METHOD PUBLIC ShiftRange : BOOL
VAR_INPUT
	StartPos	: INT;
	EndPos 		: INT;
END_VAR
VAR
	i : INT;
	N : INT := 0;
END_VAR
IF(StartPos < EndPos AND EndPos <= ArraySize) THEN
	N := EndPos - StartPos - 1;
	FOR i:= 0 TO N DO
		MEMCPY(ADR(DataRepository[EndPos-i]), ADR(DataRepository[EndPos-i-1]), SIZEOF(stShiftData));
	END_FOR;
ELSE
	; //Error;
END_IF;

// Clear start position data array
MEMSET(ADR(DataRepository[StartPos]), 16#00, SIZEOF(stShiftData));
END_METHOD

METHOD Update : BOOL
VAR_INPUT
END_VAR
// TODO: GraphQL mutation with FIFO
END_METHOD

END_FUNCTION_BLOCK

// ---- FBs/FB_PneumaticActuator_2EV.TcPOU
FUNCTION_BLOCK FB_PneumaticActuator_2EV
VAR_INPUT
	I_bEnable					: BOOL;
	I_bCmdFwd					: BOOL;					// Comando avanti
	I_bCmdBwd					: BOOL;					// Comando indietro
	I_eReadyPos					: eReadyPos := Bwd;		// Posizione iniziale di fuori ingombro per start ciclo 0=indietro, 1=avanti
	I_bSensorFwd				: BOOL;					// Sensore avanti
	I_bSensorBwd				: BOOL;					// Sensore indietro
	I_bCmdReset					: BOOL;					// Reset allarmi
	I_bAirPresence				: BOOL;					// Presenza aria nel circuito - Abilitazione comandi
	I_bManualMode				: BOOL;					// Modo manuale
	I_bEvMonostable				: BOOL;
	I_tTimeoutFwd				: TIME := T#0S;			// Timeout movimento avanti
	I_tTimeoutBwd				: TIME := T#0S;			// Timeout movimento indietro
	I_tDelaySensorFwd			: TIME := T#0S;			// Ritardo sul sensore avanti
	I_tDelaySensorBwd			: TIME := T#0S;			// Ritardo sul sensore indietro
	I_tWarningFwd				: TIME := T#0S;			// Warning movimento avanti  
	I_tWarningBwd				: TIME := T#0S;			// Warning movimento indietro
END_VAR

VAR_OUTPUT
	Q_bActuatorFwd				: BOOL := FALSE;		// Comando avanti
	Q_bActuatorBwd				: BOOL := FALSE;		// Comando indietro
	Q_bTimeoutFwd				: BOOL := FALSE;		// Timeout avanti attivo
	Q_bTimeoutBwd				: BOOL := FALSE;		// Timeout indietro attivo
	Q_bWarningFwd				: BOOL := FALSE;		// Warning avanti attivo
	Q_bWarningBwd				: BOOL := FALSE;		// Warning indietro attivo
	Q_bSensorBroken				: BOOL := FALSE;		// Timeout entrambi sensori attivi
	Q_bDelaySensorFwd			: BOOL := FALSE;		// Stato sensore avanti ritardato
	Q_bDelaySensorBwd			: BOOL := FALSE;		// Stato sensore indietro ritardato
	Q_tElapsedTimeFwd			: UINT := 0;			// Durata movimento avanti
	Q_tElapsedTimeBwd			: UINT := 0;			// Durata movimento indietro
	Q_tLastFwd					: UINT := 0;			// Durata ultimo movimento avanti
	Q_tLastBwd					: UINT := 0;			// Durata ultimo movimento indietro
	Q_bReadyPos					: BOOL := FALSE;		// In posizione iniziale di fuori ingombro
	Q_eStatus					: eEV_Status := eEV_Status.NotUsed; // Descrizione stato funzione
END_VAR

VAR
	_TON_TimerFwd				: TON;
	_TON_TimerBwd				: TON;
	_TON_WarningFwd				: TON;
	_TON_WarningBwd				: TON;
	_TON_TimerSensorBroken		: TON;
	_TON_DelaySensorFwd			: TON;	
	_TON_DelaySensorBwd			: TON;
END_VAR

_TON_DelaySensorFwd(IN := I_bSensorFwd, PT := I_tDelaySensorFwd, Q => Q_bDelaySensorFwd);					
_TON_DelaySensorBwd(IN := I_bSensorBwd, PT := I_tDelaySensorBwd, Q => Q_bDelaySensorBwd);

_TON_TimerFwd(IN := Q_bActuatorFwd AND NOT I_bSensorFwd AND I_bAirPresence);					
_TON_TimerBwd(IN := Q_bActuatorBwd AND NOT I_bSensorBwd AND I_bAirPresence);
												
IF I_bEnable THEN
	IF I_bManualMode THEN
		// Logica di movimento in indietro
		IF I_bCmdBwd THEN
			Q_bActuatorBwd := TRUE;
			Q_bActuatorFwd := FALSE;
			Q_eStatus := eEV_Status.MovingBackward;
		ELSIF NOT I_bEvMonostable AND NOT I_bCmdBwd THEN
			Q_bActuatorBwd := FALSE;
		END_IF
		// Logica di movimento in avanti
		IF I_bCmdFwd THEN
			Q_bActuatorFwd := TRUE;
			Q_bActuatorBwd := FALSE;
			Q_eStatus := eEV_Status.MovingForward;  
		ELSIF NOT I_bEvMonostable AND NOT I_bCmdFwd THEN
			Q_bActuatorFwd := FALSE;
		END_IF
	ELSE
		// Logica di movimento in avanti
		IF I_bCmdFwd AND NOT I_bSensorFwd THEN
		    Q_bActuatorFwd := TRUE;          
		    Q_bActuatorBwd := FALSE;         
		    Q_eStatus := eEV_Status.MovingForward;   
		ELSIF I_bSensorFwd AND NOT I_bEvMonostable THEN
		    Q_bActuatorFwd := FALSE;         
		END_IF
	
		// Logica di movimento indietro
		IF I_bCmdBwd AND NOT I_bSensorBwd THEN
		    Q_bActuatorBwd := TRUE;          				
		    Q_bActuatorFwd := FALSE;         				
		    Q_eStatus := eEV_Status.MovingBackward;	
		ELSIF I_bSensorBwd AND NOT I_bEvMonostable THEN
		    Q_bActuatorBwd := FALSE;         				
		END_IF
	END_IF	
END_IF

// Status
IF (Q_eStatus = eEV_Status.MovingBackward AND I_bSensorBwd) OR (Q_eStatus = eEV_Status.MovingForward AND I_bSensorFwd) THEN
	Q_eStatus := eEV_Status.MoveCompleted;
END_IF	

// Condizione di sicurezza: evitare comandi simultanei
IF I_bCmdFwd AND I_bCmdBwd THEN
    Q_bActuatorFwd := FALSE;	
    Q_bActuatorBwd := FALSE;    
END_IF
		
// Ready Position
IF(((I_eReadyPos = Bwd AND I_bSensorBwd) OR (I_eReadyPos = Fwd AND I_bSensorFwd)) AND NOT Q_bSensorBroken AND NOT Q_bTimeoutBwd AND NOT Q_bTimeoutFwd) THEN
	Q_bReadyPos := TRUE;
ELSE
	Q_bReadyPos := FALSE;
END_IF

// Elapsed Time	
Q_tElapsedTimeBwd := TIME_TO_UINT(_TON_TimerBwd.ET);
Q_tElapsedTimeFwd := TIME_TO_UINT(_TON_TimerFwd.ET);
IF I_bSensorFwd THEN
	Q_tLastFwd := Q_tElapsedTimeFwd;
ELSIF I_bSensorBwd THEN
	Q_tLastBwd := Q_tElapsedTimeBwd;
END_IF	

// Timeout
_TON_TimerBwd.PT := SEL(I_tTimeoutBwd = T#0S, I_tTimeoutBwd, T#99S);
_TON_TimerFwd.PT := SEL(I_tTimeoutFwd = T#0S, I_tTimeoutFwd, T#99S);
IF(_TON_TimerFwd.Q AND (I_tTimeoutFwd > T#0S)) AND I_bAirPresence THEN
	Q_bTimeoutFwd 	:= TRUE;
END_IF
IF(_TON_TimerBwd.Q AND (I_tTimeoutBwd > T#0S)) AND I_bAirPresence THEN
	Q_bTimeoutBwd 	:= TRUE;
END_IF

// Warning
_TON_WarningFwd(IN := Q_eStatus = eEV_Status.MovingForward AND NOT I_bSensorFwd AND I_bAirPresence, PT := I_tWarningFwd);					
_TON_WarningBwd(IN := Q_eStatus = eEV_Status.MovingBackward AND NOT I_bSensorBwd AND I_bAirPresence, PT := I_tWarningBwd);
IF I_bAirPresence THEN
	IF _TON_WarningFwd.Q AND (I_tWarningFwd > T#0S) THEN
		Q_bWarningFwd 	:= TRUE;
	ELSE
		Q_bWarningFwd 	:= FALSE;
	END_IF
	IF _TON_WarningBwd.Q AND (I_tWarningBwd > T#0S) THEN
		Q_bWarningBwd 	:= TRUE;
	ELSE
		Q_bWarningBwd 	:= FALSE;
	END_IF
END_IF

// Error - Sensor broken
_TON_TimerSensorBroken(PT := T#100MS, Q => Q_bSensorBroken);
IF I_bSensorFwd AND I_bSensorBwd  THEN
	_TON_TimerSensorBroken.IN := TRUE;
ELSE
	_TON_TimerSensorBroken.IN := FALSE;
END_IF

// Error management
IF Q_bTimeoutBwd OR Q_bTimeoutFwd OR Q_bSensorBroken THEN
	IF NOT Q_bSensorBroken THEN
		Q_eStatus := eEV_Status.Timeout;
	ELSE
		Q_eStatus := eEV_Status.Error;
	END_IF
END_IF

// Reset function
IF(I_bCmdReset) THEN
	Q_bTimeoutFwd 		:= FALSE;
	Q_bTimeoutBwd 		:= FALSE;
	Q_bSensorBroken		:= FALSE;
END_IF

END_FUNCTION_BLOCK

// ---- FBs/LaserMarker - LASIT/FC_Check_STX.TcPOU
FUNCTION FC_Check_STX : BOOL
VAR_INPUT
	I_sString : REFERENCE TO T_MaxString;
END_VAR
VAR
	stringPos	: INT;
END_VAR

stringPos := FIND(I_sString, STX);
IF stringPos <> 0 THEN
	I_sString := MID(I_sString, LEN(I_sString), stringPos+1);
	FC_Check_STX := TRUE;
ELSE
	FC_Check_STX := FALSE;
END_IF

END_FUNCTION

// ---- FCs/FC_EnumSnakeCaseToString.TcPOU
FUNCTION FC_EnumSnakeCaseToString : STRING
VAR_INPUT
	I_String	: T_MaxString; // Use TO_STRING(eNum) to convert the input enum. For empty string set enum = eNull
END_VAR
VAR
	pos			: INT;				
END_VAR

IF I_String <> 'eNull' THEN
	IF LEFT(I_String, 1) = 'e' THEN
		I_String := DELETE(I_String, 1, 1);
	END_IF
	pos := FIND(I_String, '_');
	WHILE pos <> 0 DO
		I_String := REPLACE(I_String, ' ', 1, pos);
		pos := FIND(I_String, '_');
	END_WHILE
	FC_EnumSnakeCaseToString := I_String;
ELSE
	FC_EnumSnakeCaseToString := '';
END_IF

END_FUNCTION

// ---- FCs/FC_MarkingLayoutSelection.TcPOU
FUNCTION FC_MarkingLayoutSelection : STRING(243)
VAR_INPUT
	Source	: eMarkingLayoutSource;
	Text	: STRING;
	MarkingCode : STRING(243);
	ProductName : STRING(243);
END_VAR

IF Source = eMarkingLayoutSource.ProductName THEN
	FC_MarkingLayoutSelection := ProductName;
ELSIF Source = eMarkingLayoutSource.FreeText THEN
	FC_MarkingLayoutSelection := Text;
ELSE
	FC_MarkingLayoutSelection := MarkingCode;
END_IF

END_FUNCTION

// ---- FCs/FC_OvrManagement.TcPOU
FUNCTION FC_OvrManagement : UINT
VAR_INPUT
	X_min 			: UINT;
    X_max 			: UINT;
    Y_min 			: UINT;
    Y_max 			: UINT;
	Counter			: UINT;
	SetCounterDone 	: BOOL;
END_VAR
VAR_OUTPUT
	SetCounte 		: BOOL;
	SetCounteValue 	: UINT;
END_VAR

IF NOT SetCounterDone THEN
	IF Counter < X_min THEN
		SetCounteValue := X_min;
		SetCounte := TRUE;
	ELSIF Counter > X_max THEN
		SetCounteValue := X_max;
		SetCounte := TRUE;
	ELSE
		FC_OvrManagement := (((Counter - X_min) * (Y_max - Y_min)) / (X_max - X_min) + Y_min);
	END_IF
ELSIF SetCounte THEN
	SetCounte := FALSE;
END_IF

END_FUNCTION

// ---- FCs/FC_PMCAlarmToBoolArray.TcPOU
FUNCTION FC_PMCAlarmToBoolArray : BOOL
VAR_INPUT
	RegA : POINTER TO BYTE;
END_VAR
VAR_OUTPUT
	AlarmList : ARRAY[0..CNC.NUM_MAX_STATION_ALARMS-1] OF BOOL;
END_VAR
VAR
	i : LWORD;
	j : DINT;
	reg: BYTE;
END_VAR

FOR i:= 0 TO 9 DO
	FOR j := 0 TO 7 DO
        AlarmList[(i*8) + j] := TO_BOOL(PBYTE_TO_BYTE((RegA+i)) AND SHL(1,j));
    END_FOR
END_FOR

END_FUNCTION

// ---- FCs/FC_PMCWarningToBoolArray.TcPOU
FUNCTION FC_PMCWarningToBoolArray : BOOL
VAR_INPUT
	RegA : POINTER TO BYTE;
END_VAR
VAR_OUTPUT
	WarningList : ARRAY[0..CNC.NUM_MAX_STATION_WARNINGS-1] OF BOOL;
END_VAR
VAR
	i : LWORD;
	j : DINT;
	reg: BYTE;
END_VAR

FOR i:= 0 TO 9 DO
	FOR j := 0 TO 7 DO
        WarningList[(i*8) + j] := TO_BOOL(PBYTE_TO_BYTE((RegA+i)) AND SHL(1,j));
    END_FOR
END_FOR

END_FUNCTION

// ---- FCs/FC_ProductStatusDatabase.TcPOU
FUNCTION FC_ProductStatusDatabase : eDbPiecesStatus
VAR_INPUT
	In					: STRING(50);
END_VAR

IF In = 'Completed' THEN
	FC_ProductStatusDatabase := eDbPiecesStatus.Completed;
ELSIF In = 'Scrap' THEN
	FC_ProductStatusDatabase := eDbPiecesStatus.Scrap;
ELSIF In = 'Processing' THEN
	FC_ProductStatusDatabase := eDbPiecesStatus.Processing;
ELSIF In = 'Fetched' THEN
	FC_ProductStatusDatabase := eDbPiecesStatus.Fetched;
ELSIF In = 'Undefined' THEN
	FC_ProductStatusDatabase := eDbPiecesStatus.Undefined;
ELSE
	FC_ProductStatusDatabase := eDbPiecesStatus.Undefined;
END_IF

END_FUNCTION

// ---- FCs/FC_SetPartProgramNameByID.TcPOU
FUNCTION FC_SetPartProgramNameByID : STRING
VAR_INPUT
	Id : LINT;
END_VAR
VAR
	sId : STRING;
	str : STRING(9) := 'O00000000';
END_VAR


sId := LINT_TO_STRING(id);
FC_SetPartProgramNameByID := CONCAT(LEFT(str, 9 - LEN(sId)), sId);

END_FUNCTION

// ---- FCs/FC_ToBoolArray.TcPOU
FUNCTION FC_ToBoolArray
VAR_INPUT
	RegSource : POINTER TO BYTE;
	RegDest	  : POINTER TO BOOL;
	Size : UINT;
END_VAR
VAR
	i 	: LWORD;
	j 	: DINT;
	reg : BYTE;
END_VAR

FOR i:=0 TO Size-1 DO
	FOR j:= 0 TO 7 DO
		RegDest^ := TO_BOOL(PBYTE_TO_BYTE((RegSource+i)) AND SHL (1,j));	
		RegDest := RegDest+1;
	END_FOR
END_FOR

END_FUNCTION

// ---- FCs/FC_ToByte.TcPOU
FUNCTION FC_ToByte : BOOL
VAR_INPUT
	RegSource : POINTER TO BOOL;
	RegDest	  : POINTER TO BYTE;
	Size : UINT;
END_VAR
VAR
	i 	: DINT;
	j   : DINT;
	bitIndex : INT;
	byteIndex : INT;
	temp : BYTE;
END_VAR

FOR i:=0 TO size-1 BY 8 DO
	temp := 0;
	FOR j:= 0 TO 7 DO
		IF RegSource[i+j] THEN
			temp := temp OR (SHL(1,j));
		END_IF
	END_FOR
	RegDest^ := temp;
	RegDest:=RegDest+1;
END_FOR

END_FUNCTION

// ---- FCs/FC_WIDP_TO_PPNAME.TcPOU
FUNCTION FC_WIDP_TO_PPNAME : STRING
VAR_INPUT
	WindP					: STRING;
END_VAR
VAR
	i				: INT;
	tempPPINT 		: INT;
	tempPPString	: STRING;
END_VAR

tempPPINT := LEN(WindP);
tempPPString := WindP;
IF tempPPINT < 8 THEN
	FOR i := 0 TO 7-tempPPINT DO
		tempPPString := CONCAT('0', tempPPString);
	END_FOR
END_IF
FC_WIDP_TO_PPNAME := tempPPString;

END_FUNCTION

// ---- FCs/Inc.TcPOU
FUNCTION Inc
VAR_INPUT
	In : POINTER TO DINT;
END_VAR

In^ := In^ + 1;

END_FUNCTION

// ---- FCs/Print.TcPOU
FUNCTION Print : BOOL
VAR_INPUT
	Text : T_MaxString;
	Arg	: T_MaxString;
END_VAR

ADSLOGSTR(ADSLOG_MSGTYPE_LOG, CONCAT(Text, '%s'), Arg);

END_FUNCTION

// ---- POUs/Database.TcPOU
PROGRAM Database
VAR
	i : UDINT;
	fbMSSQLCommandEvt 			: ARRAY[0..DB.MAX_NUMBER_ST] OF FB_SQLCommandEvt(sNetID := '', tTimeout := T#10S);
	fbMSSQLStoreProcedureEvt	: ARRAY[0..DB.MAX_NUMBER_ST] OF FB_SQLStoredProcedureEvt(sNetID := '', tTimeout := T#10S);
	tempfbMSSQLStoreProcedureEvt : ARRAY[0..DB.MAX_NUMBER_ST] OF POINTER TO FB_SQLStoredProcedureEvt; 
	fbMSSQLResult				: ARRAY[0..DB.MAX_NUMBER_ST] OF FB_SQLResultEvt(sNetID := '', tTimeout := T#10S);
	
	spUpdatePartLocationsAndProcessingDataParameters		: DUT_UpdatePartLocationsAndProcessingData;
	stParameterProcessingDataForHMI		: DUT_ProcessingDataForHMI;
	
	resetProcessinData						: BOOL;
	
	RTRIG_ProcessingDataExecute	 : R_TRIG;
	RTRIG_ShiftManTrigger0to1	 : R_TRIG;
	FTRIG_Running : F_TRIG;
	RTRIG_MachineEmpty	 : R_TRIG;
	RTRIG_ProcessingDataDoneError	: R_TRIG;
	
	ProcessingDataTrigger : BOOL;
	RTRIG_LogModeStateEventExecute	: R_TRIG;
	RTRIG_LogModeStateEventDoneOrError	: R_TRIG;
	LogModeStateEventTrigger	: BOOL;
	MemFirstCycle	: BOOL := FALSE;
	TempString	: STRING;
	SystemTimeSecStr	: STRING(2);
	TON_DelayLogModeStateEventTrigger : TON;
	RTRIG_GetSettingRepositoryExecute	: R_TRIG;
	RTRIG_GetSettingRepositoryDoneError	: R_TRIG;
	TON_MSSQL_spGetProcessingDataForHMIBusy : TON;
	memReq : BOOL;
	RTRIG_MesManualExecute	: R_TRIG;
	RTRIG_MesManualDoneError	: R_TRIG;
	myPeriod : TON;
	RTRIG_MyExe : R_TRIG;
	RTRIG_MyDone : R_TRIG;
	RTRIG_MyError : R_TRIG;
	myTime	: TIME := T#1S;
	myStart : BOOL;
	myVar : BOOL;
	myEnableConnection : BOOL;
	myConnected : ARRAY[1..5] OF BOOL;
END_VAR

IF _TaskInfo[MAIN.fbGetCurTaskIndex.index].FirstCycle THEN
	MemFirstCycle := TRUE;
END_IF
TempString := DT_TO_STRING(G.SystemTime);
SystemTimeSecStr := RIGHT(TempString, 2);
IF SystemTimeSecStr = '00' AND MemFirstCycle AND PRG_MSSQL_InitConnection.Connected THEN
	TON_DelayLogModeStateEventTrigger.IN := TRUE;
END_IF
TON_DelayLogModeStateEventTrigger(PT := T#500MS);
IF SystemTimeSecStr <> '00' AND LogModeStateEventTrigger AND NOT TON_DelayLogModeStateEventTrigger.IN THEN
 	LogModeStateEventTrigger := FALSE;
END_IF
IF TON_DelayLogModeStateEventTrigger.Q THEN
	LogModeStateEventTrigger := TRUE;
	TON_DelayLogModeStateEventTrigger.IN := FALSE;
END_IF



FOR i := 0 TO DB.MAX_NUMBER_ST DO
	tempfbMSSQLStoreProcedureEvt[i] := ADR(fbMSSQLStoreProcedureEvt[i]);
END_FOR

A_MSSQL();
A_MSSQL_ProcessingData();
Test();

ACTION A_MSSQL:
PRG_MSSQL_InitConnection(
						Enable			:=,
						DBID 			:= 1, 
						tRetryConn 	:= T#10S, 
						pSQLCommand1 	:= ADR(fbMSSQLCommandEvt[0]),
						pSQLCommand2 	:= ADR(fbMSSQLCommandEvt[1]),
						pSQLCommand3 	:= ADR(fbMSSQLCommandEvt[2]),
						pSQLCommand4 	:= ADR(fbMSSQLCommandEvt[3]),
						pSQLStoredProcedureEvt := tempfbMSSQLStoreProcedureEvt
						);
						 
PRG_MSSQL_spGetNextPartPLCData( Enable := PRG_MSSQL_InitConnection.Connected,
								OtherSPBusy := PRG_MSSQL_UpdatePartLocationsAndProcessingData.Busy OR PRG_MSSQL_UpdatePartLocationsAndProcessingData.Execute,
								fbSQLStoredProcedure := fbMSSQLStoreProcedureEvt[8],
								fbSQLResult := fbMSSQLResult[8],
								stPLCData := DB.stPLCData);
								
								
PRG_MSSQL_UpdatePartLocationsAndProcessingData(	Enable := PRG_MSSQL_InitConnection.Connected,
												fbSQLStoredProcedure := fbMSSQLStoreProcedureEvt[9],
												fbSQLResult := fbMSSQLResult[9],
												stProcessingData := DB.stProcessingData,
												Parameters := spUpdatePartLocationsAndProcessingDataParameters);
									
PRG_MSSQL_spGetProcessingDataForHMI( Enable := PRG_MSSQL_InitConnection.Connected,
									 Parameters := stParameterProcessingDataForHMI,
						  			 fbSQLStoredProcedure := fbMSSQLStoreProcedureEvt[10],
						  			 fbSQLResult := fbMSSQLResult[10],
									 ProcessingHMIDataLocation	=> DB.ProcessingHMIDataLocation,
									 ProcessingHMIDataViewData	=> DB.ProcessingHMIDataViewData); 
									 
IF G.MachineEmpty THEN
	MEMSET(ADR(DB.ProcessingHMIDataViewData), 0, SIZEOF(DB.ProcessingHMIDataViewData));
	MEMSET(ADR(DB.ProcessingHMIDataLocation), 0, SIZEOF(DB.ProcessingHMIDataLocation));
ELSE
	DB.ProcessingHMIDataLocation := PRG_MSSQL_spGetProcessingDataForHMI.ProcessingHMIDataLocation;
	DB.ProcessingHMIDataViewData := PRG_MSSQL_spGetProcessingDataForHMI.ProcessingHMIDataViewData;	
END_IF	

PRG_MSSQL_spCMD_AbortProduction(Enable := PRG_MSSQL_InitConnection.Connected,
						  	fbSQLStoredProcedure := fbMSSQLStoreProcedureEvt[36],
						  	fbSQLResult := fbMSSQLResult[36]);

//////////////// gestione PRG_MSSQL_spLogModeStateEvent ////////////////
RTRIG_LogModeStateEventExecute(CLK := G.OperatingModeOld <> HMI.Out.Header.OperatingMode OR G.MachineStateOld <> HMI.Out.Header.MachineState OR LogModeStateEventTrigger);		
RTRIG_LogModeStateEventDoneOrError(CLK := PRG_MSSQL_spLogModeStateEvent.Done OR PRG_MSSQL_spLogModeStateEvent.Error);
IF RTRIG_LogModeStateEventExecute.Q THEN
	PRG_MSSQL_spLogModeStateEvent.Execute := TRUE;
END_IF	
IF RTRIG_LogModeStateEventDoneOrError.Q THEN
	G.OperatingModeOld := HMI.Out.Header.OperatingMode;
	G.MachineStateOld := HMI.Out.Header.MachineState;
	PRG_MSSQL_spLogModeStateEvent.Execute := FALSE;
END_IF
			
PRG_MSSQL_spLogModeStateEvent.Parameters.EventId := -1;	
PRG_MSSQL_spLogModeStateEvent.Parameters.EventTimeStamp := G.SystemTime;	
PRG_MSSQL_spLogModeStateEvent.Parameters.EventType := 1;
PRG_MSSQL_spLogModeStateEvent.Parameters.Mode := HMI.Out.Header.OperatingMode;
PRG_MSSQL_spLogModeStateEvent.Parameters.State := HMI.Out.Header.MachineState;				
PRG_MSSQL_spLogModeStateEvent(Enable := PRG_MSSQL_InitConnection.Connected,
						  	fbSQLStoredProcedure := fbMSSQLStoreProcedureEvt[65],
						  	fbSQLResult := fbMSSQLResult[65]);
//////////////// gestione PRG_MSSQL_spLogModeStateEvent ////////////////

// usato direttemente da HMI
DB.fbGSCNextSPGetOrderInfoList(	Enable := PRG_MSSQL_InitConnection.Connected,
								Reset := G.ResetButton,
						  		fbSQLStoredProcedure := fbMSSQLStoreProcedureEvt[3],
						  		fbSQLResult := fbMSSQLResult[3],
								Error => DB.HMI_SP_Alarm[3].Error,
								ErrorID => DB.HMI_SP_Alarm[3].ErrorID); 

// usato direttemente da HMI			
DB.fbGSCNextSPAppendBatchToProductionQueue(Enable := PRG_MSSQL_InitConnection.Connected,
								Reset := G.ResetButton,
								fbSQLStoredProcedure := fbMSSQLStoreProcedureEvt[4],
								fbSQLResult := fbMSSQLResult[4],
								Error => DB.HMI_SP_Alarm[4].Error,
								ErrorID => DB.HMI_SP_Alarm[4].ErrorID);	 	 	

// usato direttemente da HMI								
DB.fbGSCNextSPUpdateBatchToProductionQueue(Enable := PRG_MSSQL_InitConnection.Connected,
								Reset := G.ResetButton,
								fbSQLStoredProcedure := fbMSSQLStoreProcedureEvt[5],
								fbSQLResult := fbMSSQLResult[5],
								Error => DB.HMI_SP_Alarm[5].Error,
								ErrorID => DB.HMI_SP_Alarm[5].ErrorID); 	 
								
// usato direttemente da HMI								
DB.fbGSCNextSPDeleteBatchToProductionQueue(Enable := PRG_MSSQL_InitConnection.Connected,
								Reset := G.ResetButton,
								fbSQLStoredProcedure := fbMSSQLStoreProcedureEvt[6],
								fbSQLResult := fbMSSQLResult[6],
								Error => DB.HMI_SP_Alarm[6].Error,
								ErrorID => DB.HMI_SP_Alarm[6].ErrorID);	 	 

 // usato direttemente da HMI
DB.fbGSCNextSPGetResourcesByType(Enable := PRG_MSSQL_InitConnection.Connected,
								Reset := G.ResetButton,
								fbSQLStoredProcedure := fbMSSQLStoreProcedureEvt[14],
								fbSQLResult := fbMSSQLResult[14],
								Error => DB.HMI_SP_Alarm[14].Error,
								ErrorID => DB.HMI_SP_Alarm[14].ErrorID);	 
	 
 // usato direttemente da HMI
DB.fbGSCNextSPGetResourcesByName(Enable := PRG_MSSQL_InitConnection.Connected,
								Reset := G.ResetButton,
								fbSQLStoredProcedure := fbMSSQLStoreProcedureEvt[15],
								fbSQLResult := fbMSSQLResult[15],
								Error => DB.HMI_SP_Alarm[15].Error,
								ErrorID => DB.HMI_SP_Alarm[15].ErrorID);	 	 	
						 		 
 // usato direttemente da HMI
DB.fbGSCNextSPSetResourcesByName(Enable := PRG_MSSQL_InitConnection.Connected,
								Reset := G.ResetButton,
								fbSQLStoredProcedure := fbMSSQLStoreProcedureEvt[16],
								Error => DB.HMI_SP_Alarm[16].Error,
								ErrorID => DB.HMI_SP_Alarm[16].ErrorID);	 	 		

 // usato direttemente da HMI
DB.fbGSCNextSPGetResourcesListByType(Enable := PRG_MSSQL_InitConnection.Connected,
								Reset := G.ResetButton,
								fbSQLStoredProcedure := fbMSSQLStoreProcedureEvt[17],
								fbSQLResult := fbMSSQLResult[17],
								Error => DB.HMI_SP_Alarm[17].Error,
								ErrorID => DB.HMI_SP_Alarm[17].ErrorID);	 	 	

 // usato direttemente da HMI
DB.fbGSCNextSPGetFormattedTablesFromSequences(Enable := PRG_MSSQL_InitConnection.Connected,
								Reset := G.ResetButton,
								fbSQLStoredProcedure := fbMSSQLStoreProcedureEvt[18],
								fbSQLResult := fbMSSQLResult[18],
								Error => DB.HMI_SP_Alarm[18].Error,
								ErrorID => DB.HMI_SP_Alarm[18].ErrorID);	 	 	

 // usato direttemente da HMI
DB.fbGSCNextSPGetOriginsFromSequence(Enable := PRG_MSSQL_InitConnection.Connected,
								Reset := G.ResetButton,
								fbSQLStoredProcedure := fbMSSQLStoreProcedureEvt[19],
								fbSQLResult := fbMSSQLResult[19],
								Error => DB.HMI_SP_Alarm[19].Error,
								ErrorID => DB.HMI_SP_Alarm[19].ErrorID);	 	 	

// usato direttemente da HMI
DB.fbGSCNextSPGetOrigins(Enable := PRG_MSSQL_InitConnection.Connected,
								Reset := G.ResetButton,
								fbSQLStoredProcedure := fbMSSQLStoreProcedureEvt[20],
						  		fbSQLResult := fbMSSQLResult[20],
								Error => DB.HMI_SP_Alarm[20].Error,
								ErrorID => DB.HMI_SP_Alarm[20].ErrorID);	 	 
											  
// usato direttemente da HMI
DB.fbGSCNextSPGetOriginsByName(	Enable := PRG_MSSQL_InitConnection.Connected,
								Reset := G.ResetButton,
								fbSQLStoredProcedure := fbMSSQLStoreProcedureEvt[21],
								fbSQLResult := fbMSSQLResult[21],
								Error => DB.HMI_SP_Alarm[21].Error,
								ErrorID => DB.HMI_SP_Alarm[21].ErrorID);	 	 	
								
// usato direttemente da HMI
DB.fbGSCNextSPGetOriginsBySide(	Enable := PRG_MSSQL_InitConnection.Connected,
								Reset := G.ResetButton,
								fbSQLStoredProcedure := fbMSSQLStoreProcedureEvt[22],
								fbSQLResult := fbMSSQLResult[22],
								Error => DB.HMI_SP_Alarm[22].Error,
								ErrorID => DB.HMI_SP_Alarm[22].ErrorID); 	 	

// usato direttemente da HMI
DB.fbGSCNextSPGetCutters(Enable := PRG_MSSQL_InitConnection.Connected,
								Reset := G.ResetButton,
								fbSQLStoredProcedure := fbMSSQLStoreProcedureEvt[23],
								fbSQLResult := fbMSSQLResult[23],
								Error => DB.HMI_SP_Alarm[23].Error,
								ErrorID => DB.HMI_SP_Alarm[23].ErrorID);	 	 	

// usato direttemente da HMI
DB.fbGSCNextSPGetCuttersByName(	Enable := PRG_MSSQL_InitConnection.Connected,
								Reset := G.ResetButton,
								fbSQLStoredProcedure := fbMSSQLStoreProcedureEvt[24],
								fbSQLResult := fbMSSQLResult[24],
								Error => DB.HMI_SP_Alarm[24].Error,
								ErrorID => DB.HMI_SP_Alarm[24].ErrorID);	 	 	

// usato direttemente da HMI
DB.fbGSCNextSPGetCuttersBySide(	Enable := PRG_MSSQL_InitConnection.Connected,
								Reset := G.ResetButton,
								fbSQLStoredProcedure := fbMSSQLStoreProcedureEvt[25],
								fbSQLResult := fbMSSQLResult[25],
								Error => DB.HMI_SP_Alarm[25].Error,
								ErrorID => DB.HMI_SP_Alarm[25].ErrorID);	 	

// usato direttemente da HMI
DB.fbGSCNextSPGetMillings(Enable := PRG_MSSQL_InitConnection.Connected,
								Reset := G.ResetButton,
								fbSQLStoredProcedure := fbMSSQLStoreProcedureEvt[26],
								fbSQLResult := fbMSSQLResult[26],
								Error => DB.HMI_SP_Alarm[26].Error,
								ErrorID => DB.HMI_SP_Alarm[26].ErrorID);	 	 		

// usato direttemente da HMI
DB.fbGSCNextSPGetMillingsByName(Enable := PRG_MSSQL_InitConnection.Connected,
								Reset := G.ResetButton,
								fbSQLStoredProcedure := fbMSSQLStoreProcedureEvt[27],
								fbSQLResult := fbMSSQLResult[27],
								Error => DB.HMI_SP_Alarm[27].Error,
								ErrorID => DB.HMI_SP_Alarm[27].ErrorID); 	 	

// usato direttemente da HMI
DB.fbGSCNextSPGetMillingsByFamilyName(Enable := PRG_MSSQL_InitConnection.Connected,
								Reset := G.ResetButton,
								fbSQLStoredProcedure := fbMSSQLStoreProcedureEvt[28],
								fbSQLResult := fbMSSQLResult[28],
								Error => DB.HMI_SP_Alarm[28].Error,
								ErrorID => DB.HMI_SP_Alarm[28].ErrorID); 	 		

// usato direttemente da HMI
DB.fbGSCNextSPGetResourcesByNameMilling(Enable := PRG_MSSQL_InitConnection.Connected,
								Reset := G.ResetButton,
								fbSQLStoredProcedure := fbMSSQLStoreProcedureEvt[29],
								fbSQLResult := fbMSSQLResult[29],
								Error => DB.HMI_SP_Alarm[29].Error,
								ErrorID => DB.HMI_SP_Alarm[29].ErrorID);	 	 
								
// usato direttemente da HMI					  
DB.fbGSCNextSPMES_GetOrderInfoList(Enable := PRG_MSSQL_InitConnection.Connected,
								Reset := G.ResetButton,
								fbSQLStoredProcedure := fbMSSQLStoreProcedureEvt[31],
								fbSQLResult := fbMSSQLResult[31],
								Error => DB.HMI_SP_Alarm[31].Error,
								ErrorID => DB.HMI_SP_Alarm[31].ErrorID);	 	 	

// usato direttemente da HMI					  
DB.fbGSCNextSPMES_GetOrderItems(Enable := PRG_MSSQL_InitConnection.Connected,
								Reset := G.ResetButton,
								fbSQLStoredProcedure := fbMSSQLStoreProcedureEvt[32],
								fbSQLResult := fbMSSQLResult[32],
								Error => DB.HMI_SP_Alarm[32].Error,
								ErrorID => DB.HMI_SP_Alarm[32].ErrorID);	 

// usato direttemente da HMI					  
DB.fbGSCNextSPGetOrderItems(Enable := PRG_MSSQL_InitConnection.Connected,
								Reset := G.ResetButton,
								fbSQLStoredProcedure := fbMSSQLStoreProcedureEvt[33],
								fbSQLResult := fbMSSQLResult[33],
								Error => DB.HMI_SP_Alarm[33].Error,
								ErrorID => DB.HMI_SP_Alarm[33].ErrorID);	 	 	

// usato direttemente da HMI								
DB.fbGSCNextSPGetBatchList[0](Enable := PRG_MSSQL_InitConnection.Connected,
								Reset := G.ResetButton,
								fbSQLStoredProcedure := fbMSSQLStoreProcedureEvt[34],
								fbSQLResult := fbMSSQLResult[34],
								Error => DB.HMI_SP_Alarm[34].Error,
								ErrorID => DB.HMI_SP_Alarm[34].ErrorID);	 	
								
// usato direttemente da HMI								
DB.fbGSCNextSPGetBatchList[1](Enable := PRG_MSSQL_InitConnection.Connected,
								Reset := G.ResetButton,
								fbSQLStoredProcedure := fbMSSQLStoreProcedureEvt[35],
								fbSQLResult := fbMSSQLResult[35],
								Error => DB.HMI_SP_Alarm[35].Error,
								ErrorID => DB.HMI_SP_Alarm[35].ErrorID);	 	 

// usato direttemente da HMI								
DB.fbGSCNextSPGetBatchHistory(Enable := PRG_MSSQL_InitConnection.Connected,
								Reset := G.ResetButton,
								fbSQLStoredProcedure := fbMSSQLStoreProcedureEvt[37],
								fbSQLResult := fbMSSQLResult[37],
								Error => DB.HMI_SP_Alarm[37].Error,
								ErrorID => DB.HMI_SP_Alarm[37].ErrorID);	 	 

// usato direttemente da HMI								
DB.fbGSCNextSPGetBatchHistoryDetail(Enable := PRG_MSSQL_InitConnection.Connected,
								Reset := G.ResetButton,
								fbSQLStoredProcedure := fbMSSQLStoreProcedureEvt[38],
								fbSQLResult := fbMSSQLResult[38],
								Error => DB.HMI_SP_Alarm[38].Error,
								ErrorID => DB.HMI_SP_Alarm[38].ErrorID); 	 

// usato direttemente da HMI									
DB.fbGSCNextSPCMD_ForceCompletedBatch(Enable := PRG_MSSQL_InitConnection.Connected,
								Reset := G.ResetButton,
								fbSQLStoredProcedure := fbMSSQLStoreProcedureEvt[39],
								fbSQLResult := fbMSSQLResult[39],
								Error => DB.HMI_SP_Alarm[39].Error,
								ErrorID => DB.HMI_SP_Alarm[39].ErrorID);	 	

// usato direttemente da HMI	
DB.fbGSCNextSPCMD_HoldBatch(Enable := PRG_MSSQL_InitConnection.Connected,
								Reset := G.ResetButton,
								fbSQLStoredProcedure := fbMSSQLStoreProcedureEvt[40],
								fbSQLResult := fbMSSQLResult[40],
								Error => DB.HMI_SP_Alarm[40].Error,
								ErrorID => DB.HMI_SP_Alarm[40].ErrorID);	  	

// usato direttemente da HMI											
DB.fbGSCNextSPCMD_RecoverBatch(Enable := PRG_MSSQL_InitConnection.Connected,
								Reset := G.ResetButton,
								fbSQLStoredProcedure := fbMSSQLStoreProcedureEvt[41],
								fbSQLResult := fbMSSQLResult[41],
								Error => DB.HMI_SP_Alarm[41].Error,
								ErrorID => DB.HMI_SP_Alarm[41].ErrorID); 	  	

// usato direttemente da HMI		
DB.fbGSCNextSPCMD_RestartBatch(Enable := PRG_MSSQL_InitConnection.Connected,
								Reset := G.ResetButton,
								fbSQLStoredProcedure := fbMSSQLStoreProcedureEvt[42],
								fbSQLResult := fbMSSQLResult[42],
								Error => DB.HMI_SP_Alarm[42].Error,
								ErrorID => DB.HMI_SP_Alarm[42].ErrorID);	  	

// usato direttemente da HMI		
DB.fbGSCNextSPCMD_ResumeBatch(Enable := PRG_MSSQL_InitConnection.Connected,
								Reset := G.ResetButton,
								fbSQLStoredProcedure := fbMSSQLStoreProcedureEvt[43],
								fbSQLResult := fbMSSQLResult[43],
								Error => DB.HMI_SP_Alarm[43].Error,
								ErrorID => DB.HMI_SP_Alarm[43].ErrorID); 	

// usato direttemente da HMI			
DB.fbGSCNextSPCMD_SuspendBatch(Enable := PRG_MSSQL_InitConnection.Connected,
								Reset := G.ResetButton,
								fbSQLStoredProcedure := fbMSSQLStoreProcedureEvt[44],
								fbSQLResult := fbMSSQLResult[44],
								Error => DB.HMI_SP_Alarm[44].Error,
								ErrorID => DB.HMI_SP_Alarm[44].ErrorID); 	  	

// usato direttemente da HMI		
DB.fbGSCNextSPCMD_UnholdBatch(Enable := PRG_MSSQL_InitConnection.Connected,
								Reset := G.ResetButton,
								fbSQLStoredProcedure := fbMSSQLStoreProcedureEvt[45],
								fbSQLResult := fbMSSQLResult[45],
								Error => DB.HMI_SP_Alarm[45].Error,
								ErrorID => DB.HMI_SP_Alarm[45].ErrorID);	 	

// usato direttemente da HMI	
RTRIG_MesManualExecute(CLK := HMI.General.Mes.PS);
RTRIG_MesManualDoneError(CLK := DB.fbGSCNextSPUpdateSettingRepositoryByName.Done OR DB.fbGSCNextSPUpdateSettingRepositoryByName.Execute);	
IF RTRIG_MesManualExecute.Q THEN
	DB.fbGSCNextSPUpdateSettingRepositoryByName.Name := 'MESEnabled';
	DB.fbGSCNextSPUpdateSettingRepositoryByName.Execute := TRUE;
	DB.fbGSCNextSPUpdateSettingRepositoryByName.JsonValue := HMI.General.Mes.Data;
END_IF			
IF RTRIG_MesManualDoneError.Q THEN
	IF DB.fbGSCNextSPUpdateSettingRepositoryByName.Done THEN
		DB.MesReadStatusCmd := TRUE;
	END_IF
	DB.fbGSCNextSPUpdateSettingRepositoryByName.Execute := FALSE;
END_IF									
DB.fbGSCNextSPUpdateSettingRepositoryByName(Enable := PRG_MSSQL_InitConnection.Connected,
								Reset := G.ResetButton,
								fbSQLStoredProcedure := fbMSSQLStoreProcedureEvt[46],
								fbSQLResult := fbMSSQLResult[46],
								Error => DB.HMI_SP_Alarm[46].Error,
								ErrorID => DB.HMI_SP_Alarm[46].ErrorID);
								
// usato direttemente da HMI								
DB.fbGSCNextSPGetSettingRepositoryList(Enable := PRG_MSSQL_InitConnection.Connected,
								Reset := G.ResetButton,
								fbSQLStoredProcedure := fbMSSQLStoreProcedureEvt[47],
								fbSQLResult := fbMSSQLResult[47],
								Error => DB.HMI_SP_Alarm[47].Error,
								ErrorID => DB.HMI_SP_Alarm[47].ErrorID);	  	

// usato direttemente da HMI								
DB.fbGSCNextSPGetBatchDetailById(Enable := PRG_MSSQL_InitConnection.Connected,
								Reset := G.ResetButton,
								fbSQLStoredProcedure := fbMSSQLStoreProcedureEvt[48],
								fbSQLResult := fbMSSQLResult[48],
								Error => DB.HMI_SP_Alarm[48].Error,
								ErrorID => DB.HMI_SP_Alarm[48].ErrorID);  

// usato direttemente da HMI								
DB.fbGSCNextSPChangeBatchPositionInProductionQueue(Enable := PRG_MSSQL_InitConnection.Connected,
								Reset := G.ResetButton,
								fbSQLStoredProcedure := fbMSSQLStoreProcedureEvt[49],
								fbSQLResult := fbMSSQLResult[49],
								Error => DB.HMI_SP_Alarm[49].Error,
								ErrorID => DB.HMI_SP_Alarm[49].ErrorID);	

// usato direttemente da HMI									
DB.fbGSCNextSPGetCuttersOnDrum(Enable := PRG_MSSQL_InitConnection.Connected,
								Reset := G.ResetButton,
								fbSQLStoredProcedure := fbMSSQLStoreProcedureEvt[50],
								fbSQLResult := fbMSSQLResult[50],
								Error => DB.HMI_SP_Alarm[50].Error,
								ErrorID => DB.HMI_SP_Alarm[50].ErrorID);

// usato direttemente da HMI	
DB.fbGSCNextSPGetCuttersComboboxFormatted(Enable := PRG_MSSQL_InitConnection.Connected,
								Reset := G.ResetButton,
								fbSQLStoredProcedure := fbMSSQLStoreProcedureEvt[51],
								fbSQLResult := fbMSSQLResult[51],
								Error => DB.HMI_SP_Alarm[51].Error,
								ErrorID => DB.HMI_SP_Alarm[51].ErrorID);	 	
								
// usato direttemente da HMI
DB.fbGSCNextSPUpdateCuttersOnDrum(Enable := PRG_MSSQL_InitConnection.Connected,
								Reset := G.ResetButton,
								fbSQLStoredProcedure := fbMSSQLStoreProcedureEvt[52],
								fbSQLResult := fbMSSQLResult[52],
								Error => DB.HMI_SP_Alarm[52].Error,
								ErrorID => DB.HMI_SP_Alarm[52].ErrorID);

// usato direttemente da HMI								
DB.fbGSCNextSPCheckCutterAlreadyPresentOnDrums(Enable := PRG_MSSQL_InitConnection.Connected,
								Reset := G.ResetButton,
								fbSQLStoredProcedure := fbMSSQLStoreProcedureEvt[53],
								fbSQLResult := fbMSSQLResult[53],
								Error => DB.HMI_SP_Alarm[53].Error,
								ErrorID => DB.HMI_SP_Alarm[53].ErrorID);
								
// usato direttemente da HMI								
DB.fbGSCNextSPUpdateCutterData(Enable := PRG_MSSQL_InitConnection.Connected,
								Reset := G.ResetButton,
								fbSQLStoredProcedure := fbMSSQLStoreProcedureEvt[54],
								fbSQLResult := fbMSSQLResult[54],
								Error => DB.HMI_SP_Alarm[54].Error,
								ErrorID => DB.HMI_SP_Alarm[54].ErrorID);	

// usato direttemente da HMI								
DB.fbGSCNextSPGetProfilesByFamilyName(Enable := PRG_MSSQL_InitConnection.Connected,
								Reset := G.ResetButton,
								fbSQLStoredProcedure := fbMSSQLStoreProcedureEvt[55],
								fbSQLResult := fbMSSQLResult[55],
								Error => DB.HMI_SP_Alarm[55].Error,
								ErrorID => DB.HMI_SP_Alarm[55].ErrorID);	
								
// usato direttemente da HMI								
DB.fbGSCNextSPGetProfiles(Enable := PRG_MSSQL_InitConnection.Connected,
								Reset := G.ResetButton,
								fbSQLStoredProcedure := fbMSSQLStoreProcedureEvt[56],
								fbSQLResult := fbMSSQLResult[56],
								Error => DB.HMI_SP_Alarm[56].Error,
								ErrorID => DB.HMI_SP_Alarm[56].ErrorID);
								
// usato direttemente da HMI
DB.fbGSCNextSPGetFamilyNamesForCombobox(Enable := PRG_MSSQL_InitConnection.Connected,
								Reset := G.ResetButton,
								fbSQLStoredProcedure := fbMSSQLStoreProcedureEvt[57],
								fbSQLResult := fbMSSQLResult[57],
								Error => DB.HMI_SP_Alarm[57].Error,
								ErrorID => DB.HMI_SP_Alarm[57].ErrorID);
								
// usato direttemente da HMI
DB.fbGSCNextSPGetCuttersFromFamilyName(Enable := PRG_MSSQL_InitConnection.Connected,
								Reset := G.ResetButton,
								fbSQLStoredProcedure := fbMSSQLStoreProcedureEvt[58],
								fbSQLResult := fbMSSQLResult[58],
								Error => DB.HMI_SP_Alarm[58].Error,
								ErrorID => DB.HMI_SP_Alarm[58].ErrorID);
								
// usato direttemente da HMI
DB.fbGSCNextSPDeleteProfile(Enable := PRG_MSSQL_InitConnection.Connected,
								Reset := G.ResetButton,
								fbSQLStoredProcedure := fbMSSQLStoreProcedureEvt[59],
								fbSQLResult := fbMSSQLResult[59],
								Error => DB.HMI_SP_Alarm[59].Error,
								ErrorID => DB.HMI_SP_Alarm[59].ErrorID);
								
// usato direttemente da HMI
DB.fbGSCNextSPAddProfile(Enable := PRG_MSSQL_InitConnection.Connected,
								Reset := G.ResetButton,
								fbSQLStoredProcedure := fbMSSQLStoreProcedureEvt[60],
								fbSQLResult := fbMSSQLResult[60],
								Error => DB.HMI_SP_Alarm[60].Error,
								ErrorID => DB.HMI_SP_Alarm[60].ErrorID);
								
// usato direttemente da HMI
DB.fbGSCNextSPDeleteCutter(Enable := PRG_MSSQL_InitConnection.Connected,
								Reset := G.ResetButton,
								fbSQLStoredProcedure := fbMSSQLStoreProcedureEvt[61],
								fbSQLResult := fbMSSQLResult[61],
								Error => DB.HMI_SP_Alarm[61].Error,
								ErrorID => DB.HMI_SP_Alarm[61].ErrorID);
								
// usato direttemente da HMI
DB.fbGSCNextSPAddCutter(Enable := PRG_MSSQL_InitConnection.Connected,
								Reset := G.ResetButton,
								fbSQLStoredProcedure := fbMSSQLStoreProcedureEvt[62],
								fbSQLResult := fbMSSQLResult[62],
								Error => DB.HMI_SP_Alarm[62].Error,
								ErrorID => DB.HMI_SP_Alarm[62].ErrorID);
								
// usato direttemente da HMI
DB.fbGSCNextSPGetBroachingProfileSettings(Enable := PRG_MSSQL_InitConnection.Connected,
								Reset := G.ResetButton,
								fbSQLStoredProcedure := fbMSSQLStoreProcedureEvt[63],
								fbSQLResult := fbMSSQLResult[63],
								Error => DB.HMI_SP_Alarm[63].Error,
								ErrorID => DB.HMI_SP_Alarm[63].ErrorID);

// usato direttemente da HMI								
DB.fbGSCNextSPUpdateBroachingProfileSettings(Enable := PRG_MSSQL_InitConnection.Connected,
								Reset := G.ResetButton,
								fbSQLStoredProcedure := fbMSSQLStoreProcedureEvt[64],
								fbSQLResult := fbMSSQLResult[64],
								Error => DB.HMI_SP_Alarm[64].Error,
								ErrorID => DB.HMI_SP_Alarm[64].ErrorID);	 
							
// fbMSSQLStoreProcedureEvt[65] usato da plc, vedi in alto

// usato direttemente da HMI	
RTRIG_GetSettingRepositoryExecute(CLK := DB.MesReadStatusCmd);	
RTRIG_GetSettingRepositoryDoneError(CLK := DB.fbGSCNextSPGetSettingRepositoryByName.Done OR DB.fbGSCNextSPGetSettingRepositoryByName.Error);	
IF RTRIG_GetSettingRepositoryExecute.Q THEN
	DB.fbGSCNextSPGetSettingRepositoryByName.Name := 'MESEnabled';
	DB.fbGSCNextSPGetSettingRepositoryByName.Execute := TRUE;
END_IF 
IF RTRIG_GetSettingRepositoryDoneError.Q THEN
	IF DB.fbGSCNextSPGetSettingRepositoryByName.Done THEN
		HMI.General.Mes.LS := DB.fbGSCNextSPGetSettingRepositoryByName.Data;
	END_IF	
	DB.MesReadStatusCmd := FALSE;
	DB.fbGSCNextSPGetSettingRepositoryByName.Execute := FALSE;
END_IF 				
DB.fbGSCNextSPGetSettingRepositoryByName(Enable := PRG_MSSQL_InitConnection.Connected,
								Reset := G.ResetButton,
								fbSQLStoredProcedure := fbMSSQLStoreProcedureEvt[66],
								fbSQLResult := fbMSSQLResult[66],
								Error => DB.HMI_SP_Alarm[66].Error,
								ErrorID => DB.HMI_SP_Alarm[66].ErrorID);
END_ACTION

ACTION A_MSSQL_ProcessingData:
IF NOT G.fbProcessingData[1].UnloadingStation THEN
	G.PMCShiftDataSlide := HMI.ShiftData[1];
END_IF
IF NOT G.fbProcessingData[2].UnloadingStation THEN
	G.PMCShiftDataLaser := HMI.ShiftData[2];
END_IF
IF NOT G.fbProcessingData[5].UnloadingStation THEN
	G.PMCShiftDataCart := HMI.ShiftData[5];
END_IF
IF NOT G.fbProcessingData[8].UnloadingStation THEN
	G.PMCShiftDataDeburring := HMI.ShiftData[8];
END_IF
IF NOT G.fbProcessingData[9].UnloadingStation THEN
	G.PMCShiftDataPallet := HMI.ShiftData[9];
END_IF
IF NOT G.fbProcessingData[14].UnloadingStation THEN
	G.PMCShiftDataPallet := HMI.ShiftData[14];
END_IF

G.fbProcessingData[0](PMCShiftManData  := HMI.ShiftData[0],
					NumStation		 := 0, 
					FirstStation	 := TRUE,
					StationOne		 := FALSE,
					UnloadingStation := FALSE,
					Trigger			 := ProcessingDataTrigger,
					stProcessingData => (*DB.stProcessingData[0]*));

G.fbProcessingData[1](PMCShiftManData  := G.PMCShiftDataSlide,
					NumStation		 := 1, 
					FirstStation	 := FALSE,
					StationOne		 := FALSE,
					Trigger			 := ProcessingDataTrigger,
					ProductStatus 	 := FC_ProductStatus(G.PMCShiftDataSlide.FLAGP),
					stProcessingData => (*DB.stProcessingData[1]*));
					
G.fbProcessingData[2](PMCShiftManData  := G.PMCShiftDataLaser,
					NumStation		 := 2, 
					FirstStation	 := FALSE,
					StationOne		 := FALSE,
					Trigger			 := ProcessingDataTrigger,
					ProductStatus 	 := FC_ProductStatus(G.PMCShiftDataLaser.FLAGP),
					stProcessingData => (*DB.stProcessingData[2]*));
					
G.fbProcessingData[3](PMCShiftManData  := HMI.ShiftData[3],
					NumStation		 := 3, 
					FirstStation	 := FALSE,
					StationOne		 := FALSE,
					UnloadingStation := FALSE,
					Trigger			 := ProcessingDataTrigger,
					ProductStatus 	 := FC_ProductStatus(HMI.ShiftData[3].FLAGP),
					stProcessingData => (*DB.stProcessingData[3]*));
					
G.fbProcessingData[4](PMCShiftManData  := HMI.ShiftData[4],
					NumStation		 := 4, 
					FirstStation	 := FALSE,
					StationOne		 := FALSE,
					UnloadingStation := FALSE,
					Trigger			 := ProcessingDataTrigger,
					ProductStatus 	 := FC_ProductStatus(HMI.ShiftData[4].FLAGP),
					stProcessingData => (*DB.stProcessingData[4]*));
					
G.fbProcessingData[5](PMCShiftManData  := G.PMCShiftDataCart,
					NumStation		 := 5, 
					FirstStation	 := FALSE,
					StationOne		 := FALSE,
					Trigger			 := ProcessingDataTrigger,
					ProductStatus 	 := FC_ProductStatus(G.PMCShiftDataCart.FLAGP),
					stProcessingData => (*DB.stProcessingData[5]*));
					
G.fbProcessingData[6](PMCShiftManData  := HMI.ShiftData[6],
					NumStation		 := 6, 
					FirstStation	 := FALSE,
					StationOne		 := FALSE,
					UnloadingStation := FALSE,
					Trigger			 := ProcessingDataTrigger,
					ProductStatus 	 := FC_ProductStatus(HMI.ShiftData[6].FLAGP),
					stProcessingData => (*DB.stProcessingData[6]*));
					
G.fbProcessingData[7](PMCShiftManData  := HMI.ShiftData[7],
					NumStation		 := 7, 
					FirstStation	 := FALSE,
					StationOne		 := FALSE,
					UnloadingStation := FALSE,
					Trigger			 := ProcessingDataTrigger,
					ProductStatus 	 := FC_ProductStatus(HMI.ShiftData[7].FLAGP),
					stProcessingData => (*DB.stProcessingData[7]*));

G.fbProcessingData[8](PMCShiftManData  := G.PMCShiftDataDeburring,
					NumStation		 := 8, 
					FirstStation	 := FALSE,
					StationOne		 := FALSE,
					Trigger			 := ProcessingDataTrigger,
					ProductStatus 	 := FC_ProductStatus(G.PMCShiftDataDeburring.FLAGP),
					stProcessingData => (*DB.stProcessingData[8]*));
					
G.fbProcessingData[9](PMCShiftManData  := G.PMCShiftDataPallet,
					NumStation		 := 9, 
					FirstStation	 := FALSE,
					StationOne		 := FALSE,
					Trigger			 := ProcessingDataTrigger,
					ProductStatus 	 := FC_ProductStatus(G.PMCShiftDataPallet.FLAGP),
					stProcessingData => (*DB.stProcessingData[9]*));

DB.fbTriggerSequencer(Delay := T#100ms);					
RTRIG_MachineEmpty(CLK := G.MachineEmpty);
FTRIG_Running(CLK := HMI.Out.Header.MachineState = eState.Running);
RTRIG_ShiftManTrigger0to1(CLK := G.MachineEmpty AND HMI.ShiftData[0].WIDP > 0);
RTRIG_ProcessingDataExecute(CLK := (DB.fbTriggerSequencer.Out (*OR RTRIG_ShiftManTrigger0to1.Q OR RTRIG_MachineEmpty.Q*) OR FTRIG_Running.Q) AND NOT PRG_MSSQL_UpdatePartLocationsAndProcessingData.Busy);

	
IF RTRIG_ProcessingDataExecute.Q THEN
	ProcessingDataTrigger := TRUE;
END_IF
		
TON_MSSQL_spGetProcessingDataForHMIBusy(IN := NOT PRG_MSSQL_spGetProcessingDataForHMI.Busy AND NOT PRG_MSSQL_spGetProcessingDataForHMI.Execute, PT := T#100MS);		
IF (ProcessingDataTrigger (*AND TON_MSSQL_spGetProcessingDataForHMIBusy.Q*)) (*OR memReq*) THEN
	FOR i := 0 TO CNC.NUM_STATIONS DO
		DB.stProcessingData[i] := G.fbProcessingData[i].stProcessingData;
	END_FOR
	PRG_MSSQL_UpdatePartLocationsAndProcessingData.Execute := TRUE;
	ProcessingDataTrigger := FALSE;
END_IF

IF ProcessingDataTrigger AND NOT TON_MSSQL_spGetProcessingDataForHMIBusy.Q AND NOT memReq THEN
	memReq := TRUE;
END_IF

IF PRG_MSSQL_UpdatePartLocationsAndProcessingData.Execute AND memReq THEN
	memReq := FALSE;
END_IF
			

RTRIG_ProcessingDataDoneError(CLK := PRG_MSSQL_UpdatePartLocationsAndProcessingData.Done OR PRG_MSSQL_UpdatePartLocationsAndProcessingData.Error, Q => DB.fbTriggerSequencer.Reset);
IF RTRIG_ProcessingDataDoneError.Q THEN
	PRG_MSSQL_UpdatePartLocationsAndProcessingData.Execute := FALSE;
	G.fbProcessingData[1].UnloadingStation := FALSE;
	G.fbProcessingData[2].UnloadingStation := FALSE;
	G.fbProcessingData[5].UnloadingStation := FALSE;
	G.fbProcessingData[8].UnloadingStation := FALSE;
	G.fbProcessingData[9].UnloadingStation := FALSE;
	G.fbProcessingData[14].UnloadingStation := FALSE;
	G.UpdatePartLocationsAndProcessingDataTrigger := FALSE;
END_IF
END_ACTION

ACTION Test:
PRG_MSSQL_InitConnection_MyTest1(
						Enable			:= myEnableConnection,
						DBID 			:= 1, 
						tRetryConn 	:= T#10S, 
						pSQLStoredProcedureEvt := ADR(fbMSSQLStoreProcedureEvt[67]),
						Connected => myConnected[1]
						);
						
PRG_MSSQL_InitConnection_MyTest2(
						Enable			:= myEnableConnection,
						DBID 			:= 1, 
						tRetryConn 	:= T#10S, 
						pSQLStoredProcedureEvt := ADR(fbMSSQLStoreProcedureEvt[68]),
						Connected => myConnected[2]
						);
						
PRG_MSSQL_InitConnection_MyTest3(
						Enable			:= myEnableConnection,
						DBID 			:= 1, 
						tRetryConn 	:= T#10S, 
						pSQLStoredProcedureEvt := ADR(fbMSSQLStoreProcedureEvt[69]),
						Connected => myConnected[3]
						);
						
PRG_MSSQL_InitConnection_MyTest4(
						Enable			:= myEnableConnection,
						DBID 			:= 1, 
						tRetryConn 	:= T#10S, 
						pSQLStoredProcedureEvt := ADR(fbMSSQLStoreProcedureEvt[70]),
						Connected => myConnected[4]
						);
						
PRG_MSSQL_InitConnection_MyTest5(
						Enable			:= myEnableConnection,
						DBID 			:= 1, 
						tRetryConn 	:= T#10S, 
						pSQLStoredProcedureEvt := ADR(fbMSSQLStoreProcedureEvt[71]),
						Connected => myConnected[5]
						);

myPeriod(IN:=myStart AND myVar, PT := myTime); 	
RTRIG_MyExe(CLK := myPeriod.Q);
RTRIG_MyDone(CLK := PRG_MSSQL_spMyTest.Done);
RTRIG_MyError(CLK := PRG_MSSQL_spMyTest.Error);
IF RTRIG_MyExe.Q AND NOT PRG_MSSQL_spMyTest.Busy THEN
	PRG_MSSQL_spMyTest.Execute := TRUE;
	myVar := FALSE;
END_IF
IF RTRIG_MyDone.Q THEN
	PRG_MSSQL_spMyTest.Execute := FALSE;
	myVar := TRUE;
END_IF
IF RTRIG_MyError.Q THEN
	PRG_MSSQL_spMyTest.Execute := FALSE;
	myVar := FALSE;	
	myStart := FALSE;
END_IF
			
PRG_MSSQL_spMyTest(	Enable := PRG_MSSQL_InitConnection.Connected,
					fbSQLStoredProcedure := fbMSSQLStoreProcedureEvt[67],
					fbSQLResult := fbMSSQLResult[67],
					fbSQLStoredProcedure1 := fbMSSQLStoreProcedureEvt[68],
					fbSQLResult1 := fbMSSQLResult[68],
					fbSQLStoredProcedure2 := fbMSSQLStoreProcedureEvt[69],
					fbSQLResult2 := fbMSSQLResult[69],
					fbSQLStoredProcedure3 := fbMSSQLStoreProcedureEvt[70],
					fbSQLResult3 := fbMSSQLResult[70],
					fbSQLStoredProcedure4 := fbMSSQLStoreProcedureEvt[71],
					fbSQLResult4 := fbMSSQLResult[71]
);
END_ACTION

END_PROGRAM
